VAR_GLOBAL CONSTANT
	///Maximum number of skillparameters
	ParameterCnt: INT := 5;
	///Maximum number of skills per Module
	SkillCnt: INT := 15;
	///Maximum number of Statevalues of one Module
	StateCnt: INT := 10;
	///Maximum number of modules
	
	
	
	ModuleCnt: INT := 10;
	///Maximum number of Tasks in Production List
	TaskCnt: INT := 30;
	///Maximum number  of offered recipes
	OfferCnt: INT := 5;
	///Maximum number of Orders in Queue
	OrderCnt: INT := 5;
	///Number of user set parameters per recipe
	UserParameterCnt: INT := 5;
	///Number of skills per task
	TaskSkillCnt: INT := 50;
END_VAR

(* stored: Version 1.1.0.1, ProductVersion 3.1.0.25
   GVL OPCConstants: Id {840706a2-48c5-43fc-8e40-1e54666a58e5} *)
